PROGRAM OP80_MAIN
VAR
	OP80_Modeselection_FB: Mode_Selection_Block1;	
//	OP80_Cycle_Time: Cycle_Time_FB;
	TP_100ms: TP;
	Pulse_100ms: BOOL;
	Times: LREAL;
	reset: BOOL;
END_VAR

// Function Calling

OP80_Manual();
OP80_AUTOSEQUENCE();
OP80_Error();
OP80_Initialization_Seq();

//MOdeselection From HMI

IF (OP80_HMI_AutoMode AND NOT OP80_HMI_ManualMOde AND NOT OP80_HMI_StepMode) THEN
		OP80_Modeselection_FB.ModeWord:=1;
	ELSIF (NOT OP80_HMI_AutoMode AND OP80_HMI_ManualMOde AND NOT OP80_HMI_StepMode) THEN
		OP80_Modeselection_FB.ModeWord:=2;
	ELSIF  (NOT OP80_HMI_AutoMode AND NOT OP80_HMI_ManualMOde AND  OP80_HMI_StepMode) THEN
		OP80_Modeselection_FB.ModeWord:=3;
    ELSE   
		OP80_Modeselection_FB.ModeWord:=0;
END_IF
OP80_Modeselection_FB(
	ModeWord:= , 
	HomeConditionOK:=OP80_HomeConditionOK , 
	OperationEnable:=OP80_AutoSelected, 
	StartPB:=OP80_HMI_Cycle_Start , 
	SafetyAndNOError:= OP80_Safety_OK, 
	ModeAck:=OP80_Mode_Ack , 
	HomingINProgress:=OP80_HomeRunning , 
	TempHomeOK:=OP80_Temp_hmeOK , 
	ResetPB:= , 
	AutoSelected=> OP80_AutoSelected, 
	ManualSelected=> OP80_ManualSelected, 
	StepSelected=>OP80_StepSelected , 
	ModeSelAck_Indication=> , 
	StatusDisplay=> , 
	AutoRunning:=OP80_AutoRunning, 
	StepRunning:=OP80_StepRunning , 
	StartEnable:=OP80_StartEnable  , 
	MachineStop:=OP80_Machine_Stop );
(*
IF OP80_AutoSelected OR OP80_ManualSelected AND NOT ( OP80_ErrorActive OR OP80_Safety_OK) THEN
	SR60_Vert_servo.bEnable:=TRUE;
ELSE
	SR60_Vert_servo.bEnable:=FALSE;
END_IF

IF OP80_GVL.SR80_Vert_servo.bAxisError OR NOT OP80_Safety_OK  THEN
	OP80_ErrorActive:=TRUE;
END_IF

IF NOT SR60_Vert_servo.bAxisHomed THEN
	SR60_Vert_servo_not_Home:=TRUE;
ELSE
	SR60_Vert_servo_not_Home:=FALSE;
END_IF
*)
	//Cycle Time Block
//	OP80_Cycle_Time(Cycle_Start_Bit:= , Pulse_100ms:=Pulse_100ms , Time_In_Sec=>Times , CT_Running=> );

	
	
	//Pulse Generation 100ms
	TP_100ms(IN:=NOT TP_100ms.Q , PT:=T#100MS , Q=>Pulse_100ms, ET=> );

END_PROGRAM

(* stored: Version 1.1.0.1, ProductVersion 3.1.4024.11
   POU OP80_MAIN: Id {cfd391fd-bb5a-45e3-a734-8fe92b975d55}, SpecialFunc None *)
